# EPICS StreamDevice protocol: source/epics/code/lightupLED/lightupLED.proto
Terminator = CR LF;

putval{
  out "%s";
}
